// TIA Portal V17 export
// export: Created 2024-06-14T09:53:54.3068579Z, ExportSetting WithDefaults, DisplayName Totally Integrated Automation Portal, DisplayVersion V17, DisplayName TIA Portal Openness, DisplayVersion V17, DisplayName TIA Portal Version Control Interface, DisplayVersion V17, DisplayName Simotion SCOUT TIA, DisplayVersion 5.4.3.0, DisplayName SINAMICS Startdrive Advanced, DisplayVersion V17 SP1 Update 1, DisplayName SINAMICS Startdrive G110M, G120, G120C, G120D, G120P, G115D, DisplayVersion V17 SP1 Update 1, DisplayName SINAMICS Startdrive G130, G150, S120, S150, SINAMICS MV, S210, DisplayVersion V17 SP1 Update 1, DisplayName STEP 7 Professional, DisplayVersion V17, DisplayName STEP 7 Safety, DisplayVersion V17, DisplayName WinCC Professional, DisplayVersion V17
TYPE "LPG_FILL_DATA_1"
// stored: IsFailsafeCompliant false
   STRUCT
      FILL_SEQ_IN : Struct
         Cyl_IN_Pos : Bool;
         Auto_Start_Seq : Bool;
         Man_Start_Seq : Bool;
         Stop_Seq : Bool;
         Start_Timeout_Sec : DInt;
         Reset_Seq : Bool;
         Cylinder_Type : Int;
         Tare_Entry_SP : Real;
      END_STRUCT;
      FILL_SEQ_OUT : Struct
         Filled_Dat : Array[1..10] of Real;
         Domestic_Cyl : Bool;
         Commercial_Cyl : Bool;
         Start_Timeout : Bool;
         Tare_Entry_Error : Bool;
         Filling_Error : Bool;
         Step_No : Int;
         Modbus_Busy : Bool;
      END_STRUCT;
   END_STRUCT;
END_TYPE
